// TIA Portal project "Effective-ladder" (V16)

(* hardware
DEVICE "S7-1200 station_1"  S7-1200 Station
   slot 0: "Telaio di montaggio_0"  S7-1200 Rack  Rack  V1.0
   slot 1: "PLC_1"  CPU 1215C AC/DC/Rly  6ES7 215-1BG40-0XB0  V4.2
*)

// ===== PLC "PLC_1"  CPU 1215C AC/DC/Rly =====

VAR_GLOBAL   // PLC tag table "Tabella delle variabili standard"
   "State 0" AT %M20.5 : Bool;
   "State 1" AT %M20.6 : Bool;
   "AuxPhotocellStatus" AT %M20.7 : Bool;
   "State 1.1" AT %M21.0 : Bool;
   "State 1.2" AT %M21.1 : Bool;
   "HallEffectSensor" AT %I1.6 : Bool;
   "Sprinkler" AT %Q1.2 : Bool;
   "ArmTriggerOut_REQ" AT %M21.2 : Bool;
   "MotorOn" AT %M21.4 : Bool;
   "ForceMotor" AT %M21.6 : Bool;
END_VAR

VAR_GLOBAL   // PLC tag table "Tabella delle variabili standard_1"
   "GripperOpenStop" AT %I0.0 : Bool;
   "GripperCounter" AT %I0.1 : Bool;
   "ArmBackStop" AT %I0.2 : Bool;
   "ArmHCounter" AT %I0.3 : Bool;
   "ArmTopStop" AT %I0.4 : Bool;
   "ArmRotationStop" AT %I0.5 : Bool;
   "RotationalEncoder" AT %ID1000 : DInt;
   "VerticalEncoder" AT %ID1004 : DInt;
   "ConnectionButton" AT %I1.2 : Bool;
   "StopButton" AT %I1.3 : Bool;
   "ResetButton" AT %I1.4 : Bool;
   "Photosensor" AT %I1.5 : Bool;
   "GripperOpen" AT %Q0.0 : Bool;
   "GripperClose" AT %Q0.1 : Bool;
   "ArmFront" AT %Q0.2 : Bool;
   "ArmBack" AT %Q0.3 : Bool;
   "ArmDown" AT %Q0.4 : Bool;
   "ArmUp" AT %Q0.5 : Bool;
   "RotationClockwise" AT %Q0.6 : Bool;
   "RotationCounterclockwise" AT %Q0.7 : Bool;
   "GreenLed" AT %Q1.0 : Bool;
   "StopConveyor" AT %Q1.1 : Bool;
   "System_Byte" AT %MB1 : Byte;
   "FirstScan" AT %M6.0 : Bool;
   "DiagStatusUpdate" AT %M6.1 : Bool;
   "AlwaysTRUE" AT %M6.2 : Bool;
   "AlwaysFALSE" AT %M6.3 : Bool;
   "RotationalCounter" AT %MW2 : UInt;
   "Clock_Byte" AT %MB0 : Byte;
   "Clock_10Hz" AT %M0.0 : Bool;
   "Clock_5Hz" AT %M0.1 : Bool;
   "Clock_2.5Hz" AT %M0.2 : Bool;
   "Clock_2Hz" AT %M0.3 : Bool;
   "Clock_1.25Hz" AT %M0.4 : Bool;
   "Clock_1Hz" AT %M0.5 : Bool;
   "Clock_0.625Hz" AT %M0.6 : Bool;
   "Clock_0.5Hz" AT %M0.7 : Bool;
   "VerticalCounter" AT %MW4 : UInt;
   "ForceReset" AT %M7.0 : Bool;
   "ResetCompleted" AT %M7.1 : Bool;
   "TCON_Req" AT %M1.0 : Bool;
   "TDIS_Req" AT %M1.1 : Bool;
   "TSEND_Req" AT %M1.2 : Bool;
   "TRCV_Req" AT %M1.3 : Bool;
   "VerticalOverCounter" AT %MW8 : Int;
   "VerticalUnderCounter" AT %MW10 : Int;
   "RotationOverCounter" AT %MW12 : Int;
   "RotationUnderCounter" AT %MW14 : Int;
   "NormalizedRotationUnderCounter" AT %MW16 : Int;
   "NormalizedVerticalUnderCounter" AT %MW18 : Int;
   "StopAll" AT %M20.1 : Bool;
   "HRegistered" AT %M20.2 : Bool;
   "RRegistered" AT %M20.3 : Bool;
   "VRegistered" AT %M20.4 : Bool;
   "Test" AT %M21.3 : Bool;
   "TESTSOCKET" AT %M21.5 : Bool;
   "AuxStop" AT %M21.7 : Bool;
END_VAR

VAR_GLOBAL CONSTANT   // PLC tag table "Tabella delle variabili standard_1"
   "Nessuno(1)" : Pip := 65535;
   "Aggiornamento automatico(1)" : Pip := 0;
   "IPP 1(1)" : Pip := 1;
   "IPP 2(1)" : Pip := 2;
   "IPP 3(1)" : Pip := 3;
   "IPP 4(1)" : Pip := 4;
   "IPP Servo OB(1)" : Pip := 32768;
   "Local~MC(1)" : Hw_SubModule := 51;
   "Local~Common(1)" : Hw_SubModule := 50;
   "Local~Device(1)" : Hw_Device := 32;
   "Local~Configuration(1)" : Hw_SubModule := 33;
   "Local~Exec(1)" : Hw_SubModule := 52;
   "Local(1)" : Hw_SubModule := 49;
   "Local~Interfaccia_PROFINET_1(1)" : Hw_Interface := 64;
   "Local~Interfaccia_PROFINET_1~Porta_1(1)" : Hw_Interface := 65;
   "Local~Interfaccia_PROFINET_1~Porta_2(1)" : Hw_Interface := 66;
   "Local~HSC_1(1)" : Hw_Hsc := 257;
   "Local~HSC_2(1)" : Hw_Hsc := 258;
   "Local~HSC_3(1)" : Hw_Hsc := 259;
   "Local~HSC_4(1)" : Hw_Hsc := 260;
   "Local~HSC_5(1)" : Hw_Hsc := 261;
   "Local~HSC_6(1)" : Hw_Hsc := 262;
   "Local~AI_2_AQ_2_1(1)" : Hw_SubModule := 263;
   "Local~DI_14_DQ_10_1(1)" : Hw_SubModule := 264;
   "Local~Pulse_1(1)" : Hw_Pwm := 265;
   "Local~Pulse_2(1)" : Hw_Pwm := 266;
   "Local~Pulse_3(1)" : Hw_Pwm := 267;
   "Local~Pulse_4(1)" : Hw_Pwm := 268;
   "OB_Main(1)" : OB_PCYCLE := 1;
END_VAR

DATA_BLOCK "Trigger_values"   // DB7
{ S7_Optimized_Access := 'FALSE' }
VERSION : 0.1
   VAR
      Trigger : Bool;
   END_VAR
BEGIN
END_DATA_BLOCK

DATA_BLOCK "Sent_values"   // DB10
{ S7_Optimized_Access := 'FALSE' }
VERSION : 0.1
   VAR
      Rotation : Int;
      Vertical : Int;
      Horizontal : Int;
      Gripper : Bool;
   END_VAR
BEGIN
END_DATA_BLOCK

DATA_BLOCK "Received_values"   // DB12
{ S7_Optimized_Access := 'FALSE' }
VERSION : 0.1
   VAR
      Rotation : Int;
      Vertical : Int;
      Horizontal : Int;
      Gripper : Bool;
   END_VAR
BEGIN
END_DATA_BLOCK

DATA_BLOCK "Obj_detect"   // DB20
{ S7_Optimized_Access := 'FALSE' }
VERSION : 0.1
   VAR
      message : String := 'START';
   END_VAR
BEGIN
END_DATA_BLOCK

// folder: System blocks/Program resources

DATA_BLOCK "ArmHCounterCTUD"   // DB3
{ S7_Optimized_Access := 'TRUE' }
AUTHOR : Simatic
FAMILY : IEC
NAME : CNTR
VERSION : 1.0
// stored: InstanceOfName IEC_COUNTER
"IEC_COUNTER"
BEGIN
END_DATA_BLOCK

DATA_BLOCK "GripperStatus"   // DB4
{ S7_Optimized_Access := 'TRUE' }
AUTHOR : Simatic
FAMILY : IEC
NAME : CNTR
VERSION : 1.0
// stored: InstanceOfName IEC_COUNTER
"IEC_COUNTER"
BEGIN
END_DATA_BLOCK

DATA_BLOCK "ArmHStatus"   // DB6
{ S7_Optimized_Access := 'TRUE' }
AUTHOR : Simatic
FAMILY : IEC
NAME : CNTR
VERSION : 1.0
// stored: InstanceOfName IEC_COUNTER
"IEC_COUNTER"
BEGIN
END_DATA_BLOCK

DATA_BLOCK "IEC_Timer_0_DB_1"   // DB8
{ S7_Optimized_Access := 'TRUE' }
AUTHOR : Simatic
FAMILY : IEC
NAME : IEC_TMR
VERSION : 1.0
// stored: InstanceOfName IEC_TIMER
"IEC_TIMER"
BEGIN
END_DATA_BLOCK

DATA_BLOCK "ArmHStatusCTUD"   // DB13
{ S7_Optimized_Access := 'TRUE' }
AUTHOR : Simatic
FAMILY : IEC
NAME : CNTR
VERSION : 1.0
// stored: InstanceOfName IEC_COUNTER
"IEC_COUNTER"
BEGIN
END_DATA_BLOCK

DATA_BLOCK "IEC_Timer_0_DB"   // DB14
{ S7_Optimized_Access := 'TRUE' }
AUTHOR : Simatic
FAMILY : IEC
NAME : IEC_TMR
VERSION : 1.0
// stored: InstanceOfName IEC_TIMER
"IEC_TIMER"
BEGIN
END_DATA_BLOCK

DATA_BLOCK "IECTimer_0_DB1"   // DB15
{ S7_Optimized_Access := 'TRUE' }
AUTHOR : Simatic
FAMILY : IEC
NAME : IEC_TMR
VERSION : 1.0
// stored: InstanceOfName IEC_TIMER
"IEC_TIMER"
BEGIN
END_DATA_BLOCK

DATA_BLOCK "Sensor_socket_DB"   // DB17
{ S7_Optimized_Access := 'TRUE' }
AUTHOR : SIMATIC
FAMILY : MC7Plus
NAME : TC_IP_v4
VERSION : 1.0
// stored: InstanceOfName TCON_IP_v4
"TCON_IP_v4"
BEGIN
   ID := 2;
   InterfaceId := 64;
   RemotePort := 2001;
   ActiveEstablished := true;
   RemoteAddress.ADDR[1] := 192;
   RemoteAddress.ADDR[2] := 168;
   RemoteAddress.ADDR[4] := 241;
END_DATA_BLOCK

DATA_BLOCK "PLC_1_Connection_DB"   // DB21
{ S7_Optimized_Access := 'TRUE' }
AUTHOR : SIMATIC
FAMILY : MC7Plus
NAME : TC_IP_v4
VERSION : 1.0
// stored: InstanceOfName TCON_IP_v4
"TCON_IP_v4"
BEGIN
   ID := 1;
   InterfaceId := 64;
   RemotePort := 2000;
   ActiveEstablished := true;
   RemoteAddress.ADDR[1] := 192;
   RemoteAddress.ADDR[2] := 168;
   RemoteAddress.ADDR[4] := 241;
END_DATA_BLOCK

DATA_BLOCK "CONTATORE"   // DB23
{ S7_Optimized_Access := 'TRUE' }
AUTHOR : Simatic
FAMILY : IEC
NAME : CNTR
VERSION : 1.0
// stored: InstanceOfName IEC_COUNTER
"IEC_COUNTER"
BEGIN
END_DATA_BLOCK

DATA_BLOCK "IEC_Timer_0_DB_5"   // DB24
{ S7_Optimized_Access := 'TRUE' }
AUTHOR : Simatic
FAMILY : IEC
NAME : IEC_TMR
VERSION : 1.0
// stored: InstanceOfName IEC_TIMER
"IEC_TIMER"
BEGIN
END_DATA_BLOCK

DATA_BLOCK "TimerSprinkler"   // DB27
{ S7_Optimized_Access := 'TRUE' }
AUTHOR : Simatic
FAMILY : IEC
NAME : IEC_TMR
VERSION : 1.0
// stored: InstanceOfName IEC_TIMER
"IEC_TIMER"
BEGIN
END_DATA_BLOCK

// folder: (top level)

ORGANIZATION_BLOCK "Main"   // OB1, LAD, ProgramCycle
TITLE = "Main Program Sweep (Cycle)"
{ S7_Optimized_Access := 'TRUE' }
VERSION : 0.1
   VAR_INPUT
      Initial_Call : Bool;   // Initial call of this OB
      Remanence : Bool;   // =True, if remanent data are available
   END_VAR
   VAR_TEMP   // added for the SCL form of the ladder/FBD networks
      _w1 : Bool;
      _w2 : Bool;
      _w3 : Bool;
   END_VAR
BEGIN

REGION Network 1: Gestione braccio robotico
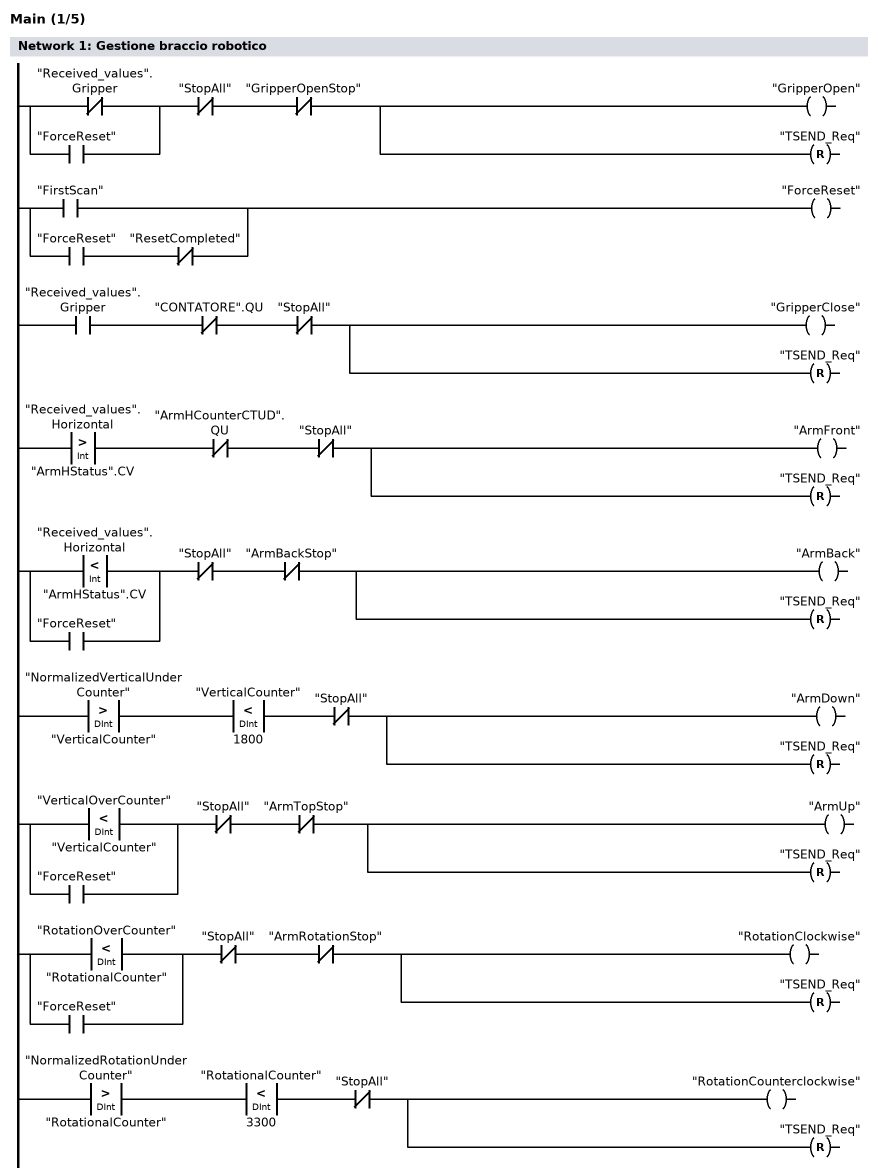
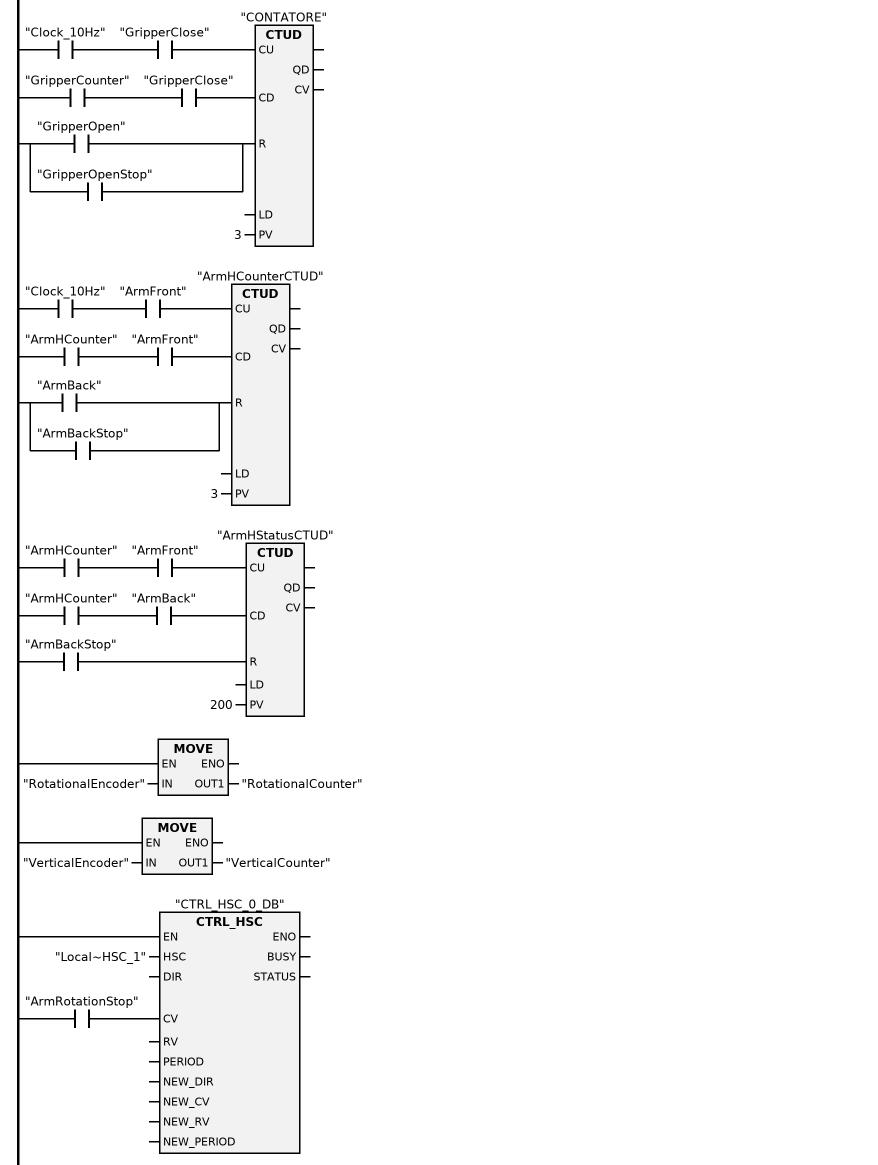
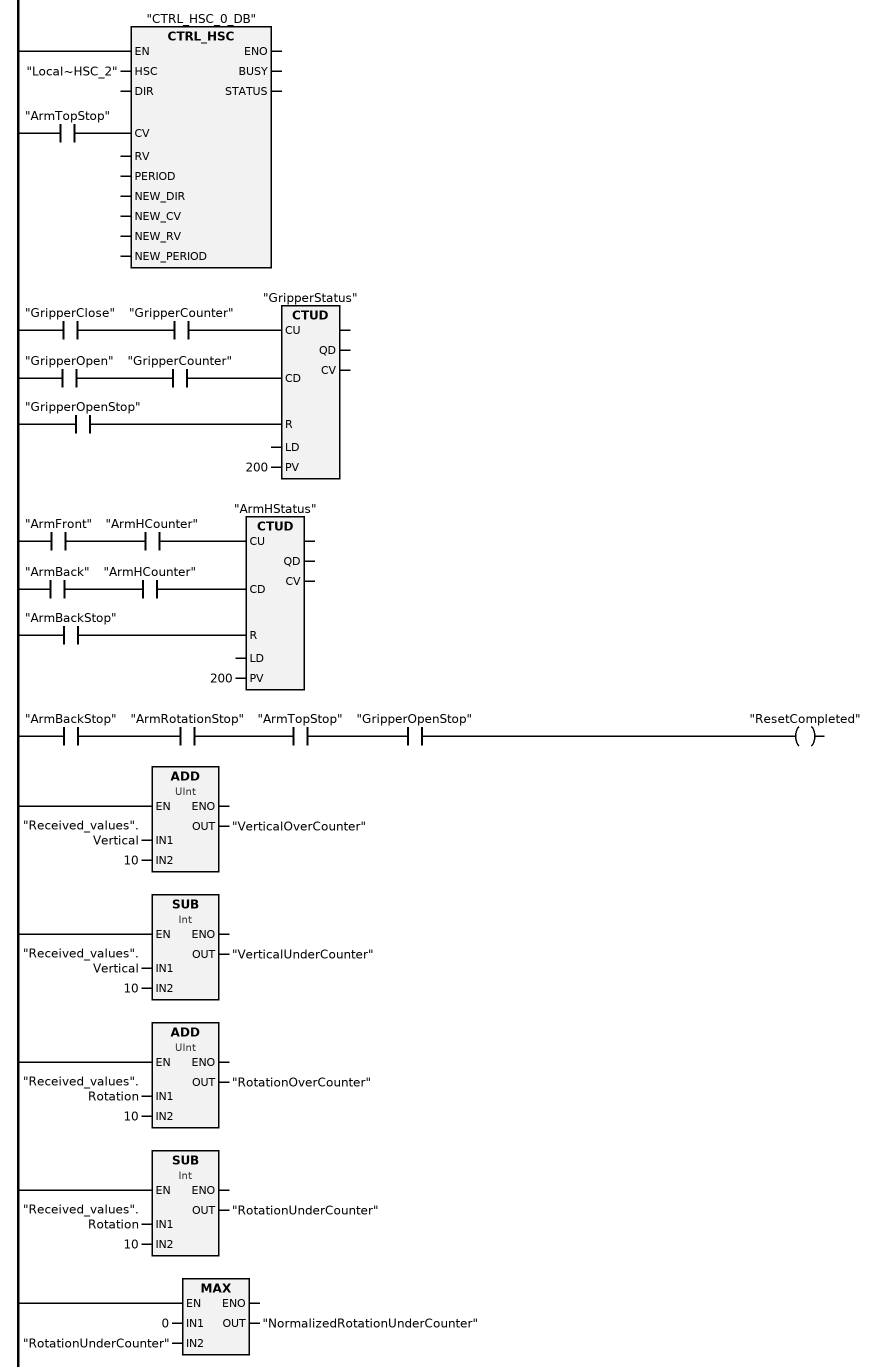
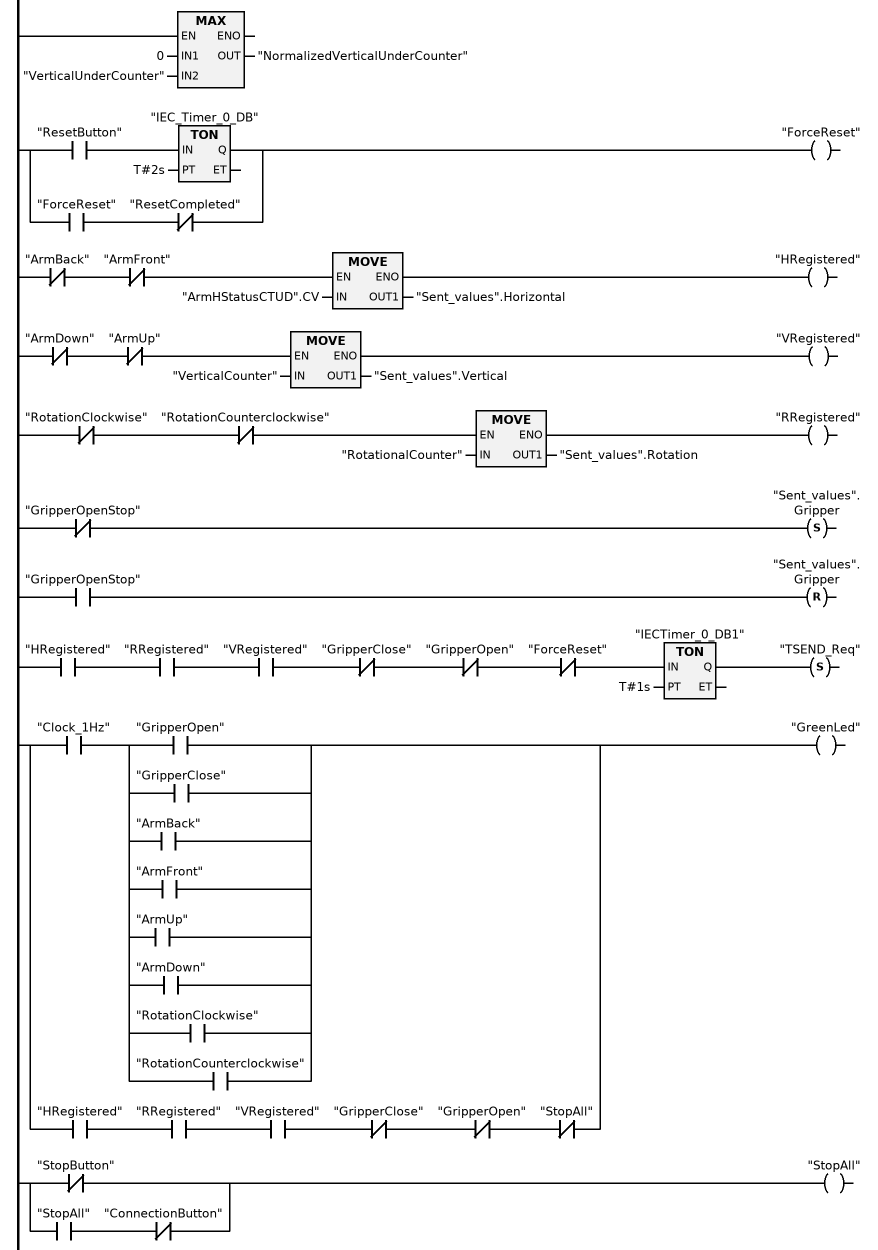
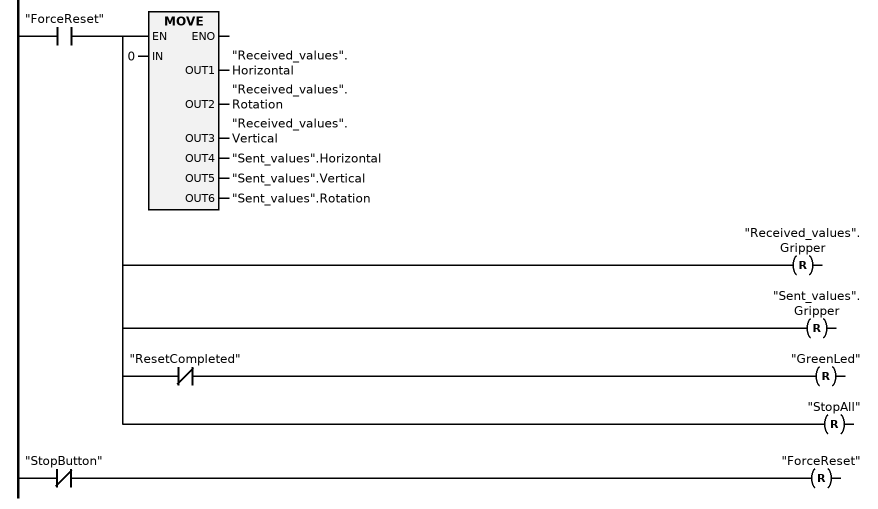
   "GripperOpen" := (NOT "Received_values".Gripper OR "ForceReset") AND NOT "StopAll" AND NOT "GripperOpenStop";
   IF "GripperOpen" THEN "TSEND_Req" := FALSE; END_IF;
   "ForceReset" := "FirstScan" OR ("ForceReset" AND NOT "ResetCompleted");
   "GripperClose" := "Received_values".Gripper AND NOT "CONTATORE".QU AND NOT "StopAll";
   IF "GripperClose" THEN "TSEND_Req" := FALSE; END_IF;
   "ArmFront" := ("Received_values".Horizontal > "ArmHStatus".CV) AND NOT "ArmHCounterCTUD".QU AND NOT "StopAll";
   IF "ArmFront" THEN "TSEND_Req" := FALSE; END_IF;
   "ArmBack" := (("Received_values".Horizontal < "ArmHStatus".CV) OR "ForceReset") AND NOT "StopAll" AND NOT "ArmBackStop";
   IF "ArmBack" THEN "TSEND_Req" := FALSE; END_IF;
   "ArmDown" := ("NormalizedVerticalUnderCounter" > "VerticalCounter") AND ("VerticalCounter" < 1800) AND NOT "StopAll";
   IF "ArmDown" THEN "TSEND_Req" := FALSE; END_IF;
   "ArmUp" := (("VerticalOverCounter" < "VerticalCounter") OR "ForceReset") AND NOT "StopAll" AND NOT "ArmTopStop";
   IF "ArmUp" THEN "TSEND_Req" := FALSE; END_IF;
   "RotationClockwise" := (("RotationOverCounter" < "RotationalCounter") OR "ForceReset") AND NOT "StopAll" AND NOT "ArmRotationStop";
   IF "RotationClockwise" THEN "TSEND_Req" := FALSE; END_IF;
   "RotationCounterclockwise" := ("NormalizedRotationUnderCounter" > "RotationalCounter") AND ("RotationalCounter" < 3300) AND NOT "StopAll";
   IF "RotationCounterclockwise" THEN "TSEND_Req" := FALSE; END_IF;
   "CONTATORE".CTUD(CU := "Clock_10Hz" AND "GripperClose",
                    CD := "GripperCounter" AND "GripperClose",
                    R := "GripperOpen" OR "GripperOpenStop",
                    PV := 3);
   "ArmHCounterCTUD".CTUD(CU := "Clock_10Hz" AND "ArmFront",
                          CD := "ArmHCounter" AND "ArmFront",
                          R := "ArmBack" OR "ArmBackStop",
                          PV := 3);
   "ArmHStatusCTUD".CTUD(CU := "ArmHCounter" AND "ArmFront",
                         CD := "ArmHCounter" AND "ArmBack",
                         R := "ArmBackStop",
                         PV := 200);
   "RotationalCounter" := "RotationalEncoder";
   "VerticalCounter" := "VerticalEncoder";
   "CTRL_HSC_0_DB"(HSC := "Local~HSC_1", CV := "ArmRotationStop");   // CTRL_HSC
   "CTRL_HSC_0_DB"(HSC := "Local~HSC_2", CV := "ArmTopStop");   // CTRL_HSC
   "GripperStatus".CTUD(CU := "GripperClose" AND "GripperCounter",
                        CD := "GripperOpen" AND "GripperCounter",
                        R := "GripperOpenStop",
                        PV := 200);
   "ArmHStatus".CTUD(CU := "ArmFront" AND "ArmHCounter",
                     CD := "ArmBack" AND "ArmHCounter",
                     R := "ArmBackStop",
                     PV := 200);
   "ResetCompleted" := "ArmBackStop" AND "ArmRotationStop" AND "ArmTopStop" AND "GripperOpenStop";
   "VerticalOverCounter" := "Received_values".Vertical + 10;
   "VerticalUnderCounter" := "Received_values".Vertical - 10;
   "RotationOverCounter" := "Received_values".Rotation + 10;
   "RotationUnderCounter" := "Received_values".Rotation - 10;
   "NormalizedRotationUnderCounter" := MAX(IN1 := 0, IN2 := "RotationUnderCounter");
   "NormalizedVerticalUnderCounter" := MAX(IN1 := 0, IN2 := "VerticalUnderCounter");
   "IEC_Timer_0_DB".TON(IN := "ResetButton", PT := T#2s);
   "ForceReset" := "IEC_Timer_0_DB".Q OR ("ForceReset" AND NOT "ResetCompleted");
   #_w1 := NOT "ArmBack" AND NOT "ArmFront";
   IF #_w1 THEN "Sent_values".Horizontal := "ArmHStatusCTUD".CV; END_IF;
   "HRegistered" := #_w1;
   #_w2 := NOT "ArmDown" AND NOT "ArmUp";
   IF #_w2 THEN "Sent_values".Vertical := "VerticalCounter"; END_IF;
   "VRegistered" := #_w2;
   #_w3 := NOT "RotationClockwise" AND NOT "RotationCounterclockwise";
   IF #_w3 THEN "Sent_values".Rotation := "RotationalCounter"; END_IF;
   "RRegistered" := #_w3;
   IF NOT "GripperOpenStop" THEN "Sent_values".Gripper := TRUE; END_IF;
   IF "GripperOpenStop" THEN "Sent_values".Gripper := FALSE; END_IF;
   "IECTimer_0_DB1".TON(IN := "HRegistered" AND "RRegistered" AND "VRegistered" AND NOT "GripperClose" AND NOT "GripperOpen" AND NOT "ForceReset",
                        PT := T#1s);
   IF "IECTimer_0_DB1".Q THEN "TSEND_Req" := TRUE; END_IF;
   "GreenLed" := ("Clock_1Hz" AND ("GripperOpen" OR "GripperClose" OR "ArmBack" OR "ArmFront" OR "ArmUp" OR "ArmDown" OR "RotationClockwise" OR "RotationCounterclockwise")) OR ("HRegistered" AND "RRegistered" AND "VRegistered" AND NOT "GripperClose" AND NOT "GripperOpen" AND NOT "StopAll");
   "StopAll" := NOT "StopButton" OR ("StopAll" AND NOT "ConnectionButton");
   IF "ForceReset" THEN
       "Received_values".Horizontal := 0;
       "Received_values".Rotation := 0;
       "Received_values".Vertical := 0;
       "Sent_values".Horizontal := 0;
       "Sent_values".Vertical := 0;
       "Sent_values".Rotation := 0;
       "Received_values".Gripper := FALSE;
       "Sent_values".Gripper := FALSE;
   END_IF;
   IF "ForceReset" AND NOT "ResetCompleted" THEN "GreenLed" := FALSE; END_IF;
   IF "ForceReset" THEN "StopAll" := FALSE; END_IF;
   IF NOT "StopButton" THEN "ForceReset" := FALSE; END_IF;
END_REGION

REGION Network 2
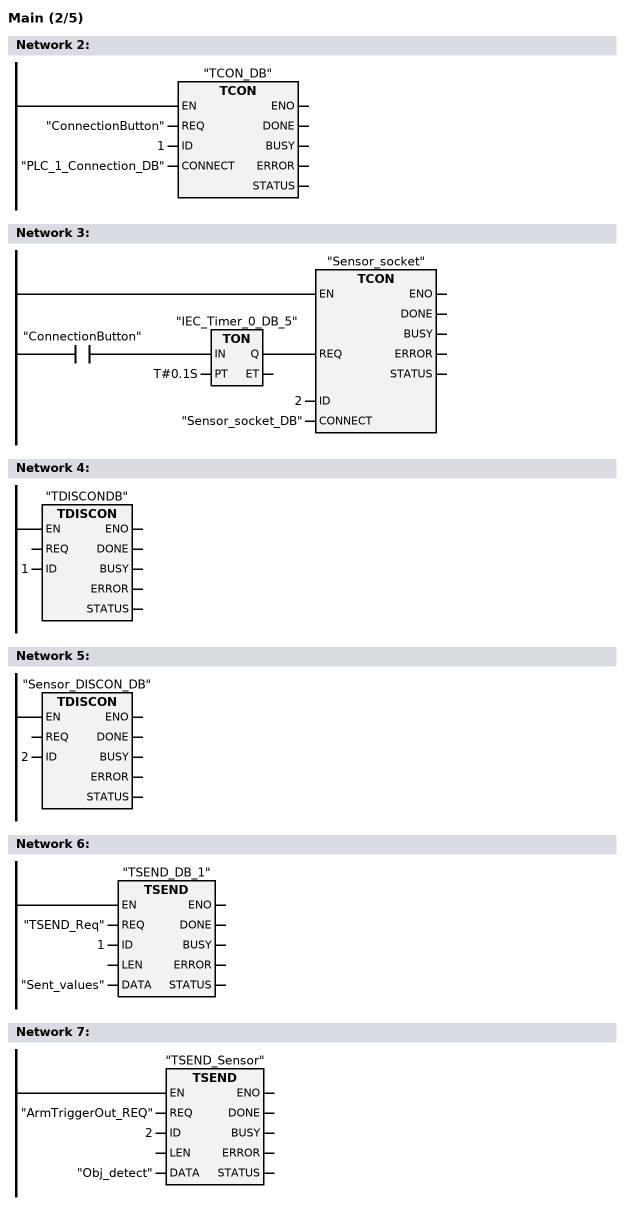
   "TCON_DB"(REQ := "ConnectionButton", ID := 1, CONNECT := "PLC_1_Connection_DB");   // TCON
END_REGION

REGION Network 3
   "IEC_Timer_0_DB_5".TON(IN := "ConnectionButton", PT := T#0.1S);
   "Sensor_socket"(REQ := "IEC_Timer_0_DB_5".Q, ID := 2, CONNECT := "Sensor_socket_DB");   // TCON
END_REGION

REGION Network 4
   "TDISCONDB"(ID := 1);   // TDISCON
END_REGION

REGION Network 5
   "Sensor_DISCON_DB"(ID := 2);   // TDISCON
END_REGION

REGION Network 6
   "TSEND_DB_1"(REQ := "TSEND_Req", ID := 1, DATA := "Sent_values");   // TSEND
END_REGION

REGION Network 7
   "TSEND_Sensor"(REQ := "ArmTriggerOut_REQ", ID := 2, DATA := "Obj_detect");   // TSEND
END_REGION

REGION Network 8
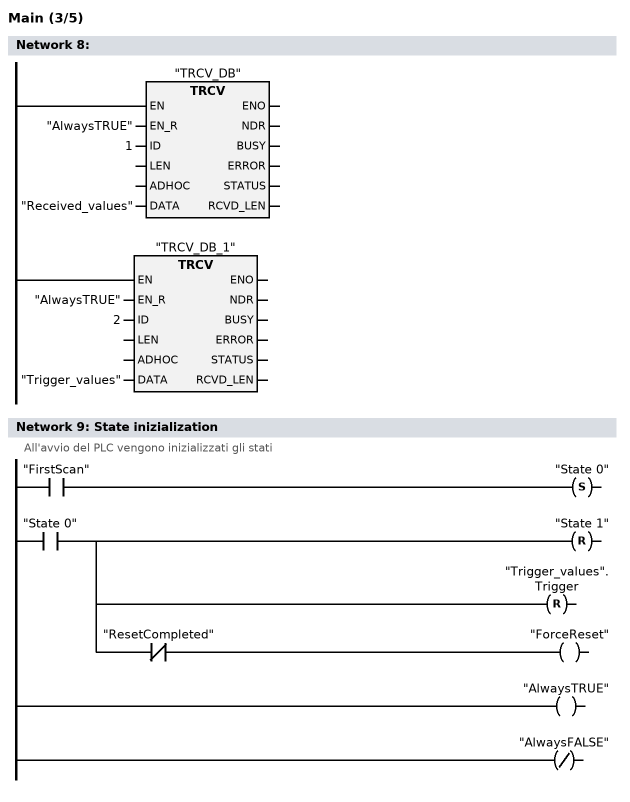
   "TRCV_DB"(EN_R := "AlwaysTRUE", ID := 1, DATA := "Received_values");   // TRCV
   "TRCV_DB_1"(EN_R := "AlwaysTRUE", ID := 2, DATA := "Trigger_values");   // TRCV
END_REGION

REGION Network 9: State inizialization
   // All'avvio del PLC vengono inizializzati gli stati
   RUNG wire#powerrail
      Contact( "FirstScan" )
      S_Coil( "State 0" )
   END_RUNG
   RUNG wire#powerrail
      Contact( "State 0" )
      wire#w1
      R_Coil( "State 1" )
   END_RUNG
   RUNG wire#w1
      R_Coil( "Trigger_values".Trigger )
   END_RUNG
   RUNG wire#w1
      I_Contact( "ResetCompleted" )
      Coil( "ForceReset" )
   END_RUNG
   RUNG wire#powerrail
      Coil( "AlwaysTRUE" )
   END_RUNG
   RUNG wire#powerrail
      I_Coil( "AlwaysFALSE" )
   END_RUNG
   // the same network as SCL:
   IF "FirstScan" THEN "State 0" := TRUE; END_IF;
   IF "State 0" THEN
       "State 1" := FALSE;
       "Trigger_values".Trigger := FALSE;
   END_IF;
   "ForceReset" := "State 0" AND NOT "ResetCompleted";
   "AlwaysTRUE" := TRUE;
   "AlwaysFALSE" := NOT TRUE;
END_REGION

REGION Network 10: State transition
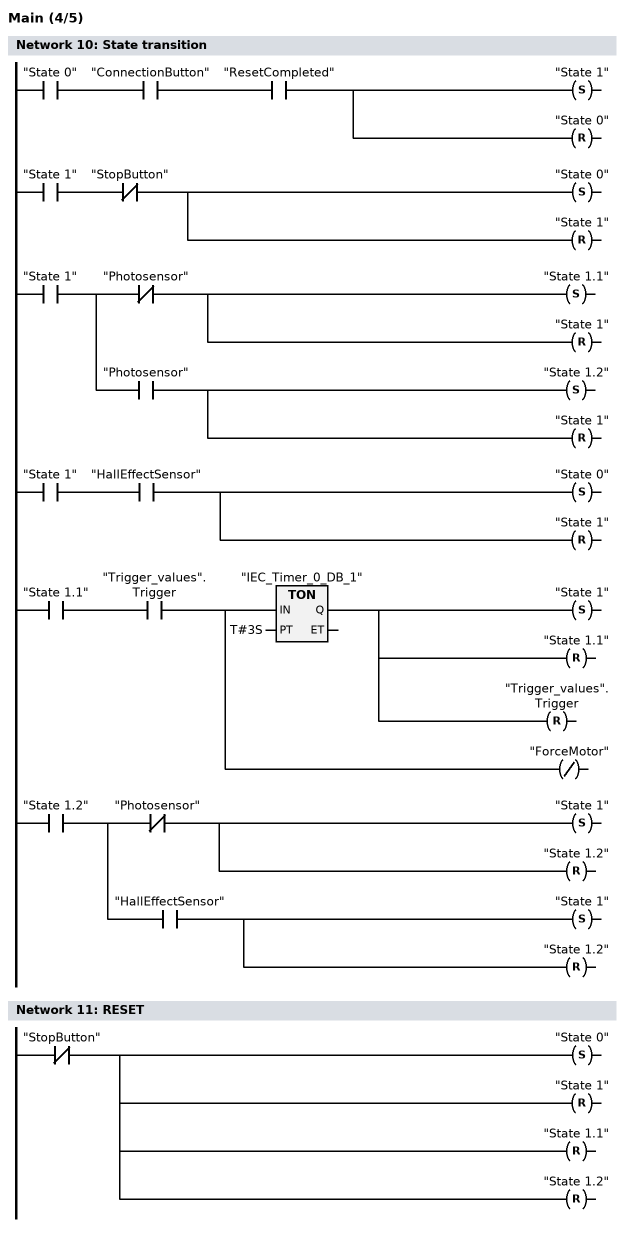
   IF "State 0" AND "ConnectionButton" AND "ResetCompleted" THEN
       "State 1" := TRUE;
       "State 0" := FALSE;
   END_IF;
   IF "State 1" AND NOT "StopButton" THEN
       "State 0" := TRUE;
       "State 1" := FALSE;
   END_IF;
   IF "State 1" AND NOT "Photosensor" THEN "State 1.1" := TRUE; END_IF;
   #_w1 := "State 1";
   IF "State 1" AND NOT "Photosensor" THEN "State 1" := FALSE; END_IF;
   IF #_w1 AND "Photosensor" THEN
       "State 1.2" := TRUE;
       "State 1" := FALSE;
   END_IF;
   IF "State 1" AND "HallEffectSensor" THEN
       "State 0" := TRUE;
       "State 1" := FALSE;
   END_IF;
   #_w2 := "State 1.1" AND "Trigger_values".Trigger;
   "IEC_Timer_0_DB_1".TON(IN := #_w2, PT := T#3S);
   IF "IEC_Timer_0_DB_1".Q THEN
       "State 1" := TRUE;
       "State 1.1" := FALSE;
       "Trigger_values".Trigger := FALSE;
   END_IF;
   "ForceMotor" := NOT #_w2;
   IF "State 1.2" AND NOT "Photosensor" THEN "State 1" := TRUE; END_IF;
   #_w3 := "State 1.2";
   IF "State 1.2" AND NOT "Photosensor" THEN "State 1.2" := FALSE; END_IF;
   IF #_w3 AND "HallEffectSensor" THEN
       "State 1" := TRUE;
       "State 1.2" := FALSE;
   END_IF;
END_REGION

REGION Network 11: RESET
   RUNG wire#powerrail
      I_Contact( "StopButton" )
      wire#w1
      S_Coil( "State 0" )
   END_RUNG
   RUNG wire#w1
      R_Coil( "State 1" )
   END_RUNG
   RUNG wire#w1
      R_Coil( "State 1.1" )
   END_RUNG
   RUNG wire#w1
      R_Coil( "State 1.2" )
   END_RUNG
   // the same network as SCL:
   IF NOT "StopButton" THEN
       "State 0" := TRUE;
       "State 1" := FALSE;
       "State 1.1" := FALSE;
       "State 1.2" := FALSE;
   END_IF;
END_REGION

REGION Network 12: Attuatori
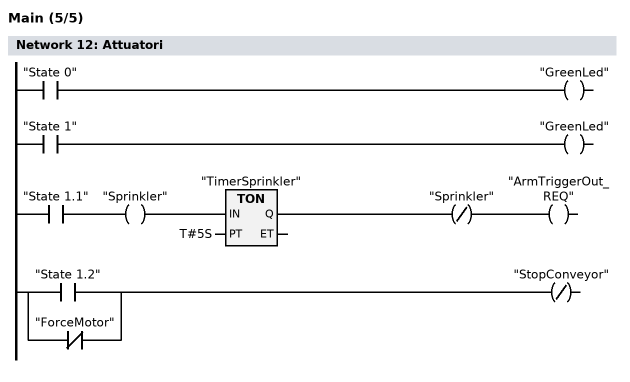
   "GreenLed" := "State 0";
   "GreenLed" := "State 1";
   "Sprinkler" := "State 1.1";
   "TimerSprinkler".TON(IN := "State 1.1", PT := T#5S);
   "Sprinkler" := NOT "TimerSprinkler".Q;
   "ArmTriggerOut_REQ" := "TimerSprinkler".Q;
   "StopConveyor" := NOT ("State 1.2" OR NOT "ForceMotor");
END_REGION
END_ORGANIZATION_BLOCK